// in the system event log; without it the behaviour is unstated.

//

// %s is filled by strArg. Passing the line as the FORMAT string instead would let
// a test label containing a percent sign corrupt the output - or worse.
ADSLOGSTR(msgCtrlMask := Severity OR ADSLOG_MSGTYPE_LOG OR ADSLOG_MSGTYPE_STRING, msgFmtStr := CONCAT(_Prefix, '%s'), strArg := Line);
_LinesWritten := _LinesWritten + 1;
END_METHOD

PROPERTY ErrorsLogged : UDINT
GET
ErrorsLogged := _ErrorsLogged;
END_GET
END_PROPERTY

PROPERTY FailuresLogged : UDINT
GET
FailuresLogged := _FailuresLogged;
END_GET
END_PROPERTY

METHOD FrameworkError
VAR_INPUT
	Source	: T_MaxString;
	Message : T_MaxString;
END_VAR
_FrameworkErrorsLogged := _FrameworkErrorsLogged + 1;

// Always an error, and never silent. This is the framework saying it could not do

// something - a rejected registration, a teardown that overran, a document that

// could not be written - and none of those is a test result.
THIS^.Emit(ADSLOG_MSGTYPE_ERROR, CONCAT(CONCAT('FRAMEWORK ', Source), CONCAT(': ', Message)));
END_METHOD

PROPERTY FrameworkErrorsLogged : UDINT
GET
FrameworkErrorsLogged := _FrameworkErrorsLogged;
END_GET
END_PROPERTY

// Always TRUE. ADSLOGSTR completes within the call, so this sink never holds a

// run open - which is precisely why it is the one to attach first.
PROPERTY IsIdle : BOOL
GET
IsIdle := TRUE;
END_GET
END_PROPERTY

// Every line this sink has written. Assert it in CI if the log is the artifact.
PROPERTY LinesWritten : UDINT
GET
LinesWritten := _LinesWritten;
END_GET
END_PROPERTY

METHOD RunFinished
VAR_INPUT
	Status	   : I_TestRunStatus;
	TargetInfo : T_MaxString;
END_VAR

VAR
	Line : T_MaxString;
END_VAR
IF Status = 0 THEN
	RETURN;
END_IF

// TargetInfo identifies where the run happened. Without it a matrix run across

// several targets produces log output that cannot be told apart.
Line := CONCAT(CONCAT(THIS^.Tally(Status), '  on '), TargetInfo);
THIS^.Emit(ADSLOG_MSGTYPE_HINT, _Rule);
// Severity follows the outcome. A log filtered to errors still shows the closing

// line of a run that went red, and shows nothing of one that did not.
//

// The same four banners, at the same severities, as the suite line. Skipped is

// not red, so it is not logged as an error; Errored is kept apart from Failed

// because nothing about the code was shown, and the reader should look elsewhere.
IF Status.Outcome = E_RunOutcome.Passed THEN
	THIS^.Emit(ADSLOG_MSGTYPE_HINT, CONCAT('===  RUN PASSED  ', Line));
ELSIF Status.Outcome = E_RunOutcome.Skipped THEN
	THIS^.Emit(ADSLOG_MSGTYPE_HINT, CONCAT('===  RUN SKIPPED ', Line));
ELSIF Status.Outcome = E_RunOutcome.Errored THEN
	THIS^.Emit(ADSLOG_MSGTYPE_ERROR, CONCAT('===  RUN ERRORED ', Line));
ELSE
	THIS^.Emit(ADSLOG_MSGTYPE_ERROR, CONCAT('===  RUN FAILED  ', Line));
END_IF

THIS^.Emit(ADSLOG_MSGTYPE_HINT, _Rule);
END_METHOD

// Opens the run with a banner, so everything between it and the closing rule

// belongs to this run and nothing else.

//

// The TwinCAT log is shared - a machine writes to it too - and test output is

// interleaved with whatever else is happening. Without a marker at BOTH ends, a

// reader scrolling back cannot tell where the run began; the failures stream

// during it and the summary only arrives at the end.
METHOD RunStarted
VAR_INPUT
	Label	   : T_MaxString;
	TargetInfo : T_MaxString;
END_VAR

VAR
	Line : T_MaxString;
END_VAR
THIS^.Emit(ADSLOG_MSGTYPE_HINT, _Rule);
Line := CONCAT('===  TEST RUN  ', Label);
IF TargetInfo <> '' THEN
	Line := CONCAT(Line, CONCAT('  on ', TargetInfo));
END_IF

THIS^.Emit(ADSLOG_MSGTYPE_HINT, Line);
THIS^.Emit(ADSLOG_MSGTYPE_HINT, _Rule);
END_METHOD

// Prepended to every line. Useful when several runs share one log - a rig

// running unit and integration suites, or a matrix across targets.
METHOD SetPrefix
VAR_INPUT
	Prefix : T_MaxString;
END_VAR
_Prefix := Prefix;
END_METHOD

// Which results reach the log. Default: failures and errors only.

//

// A suite of eighty passing tests writing eighty log lines buries the two that

// matter. Passes are counted, not narrated - the counts are already available

// through I_TestRunStatus for anyone who wants them.
METHOD SetVerbosity
VAR_INPUT
	// TRUE also logs a line for every passing and skipped test.
	IncludePasses : BOOL;
END_VAR
_IncludePasses := IncludePasses;
END_METHOD

METHOD SuiteFinished
VAR_INPUT
	Status : I_TestRunStatus;
END_VAR

VAR
	Line : T_MaxString;
END_VAR
IF Status = 0 THEN
	RETURN;
END_IF

_SuitesSeen := _SuitesSeen + 1;
Line		:= CONCAT(CONCAT(Status.Label, ': '), THIS^.Tally(Status));
// Severity follows the outcome, so a log filtered to errors still shows which

// suite was responsible rather than only the individual failures.
IF Status.Outcome = E_RunOutcome.Passed THEN
	THIS^.Emit(ADSLOG_MSGTYPE_HINT, CONCAT('SUITE PASSED  ', Line));
ELSIF Status.Outcome = E_RunOutcome.Skipped THEN
	THIS^.Emit(ADSLOG_MSGTYPE_HINT, CONCAT('SUITE SKIPPED ', Line));
ELSIF Status.Outcome = E_RunOutcome.Errored THEN
	THIS^.Emit(ADSLOG_MSGTYPE_ERROR, CONCAT('SUITE ERRORED ', Line));
ELSE
	THIS^.Emit(ADSLOG_MSGTYPE_ERROR, CONCAT('SUITE FAILED  ', Line));
END_IF
END_METHOD

PROPERTY SuitesSeen : UDINT
GET
SuitesSeen := _SuitesSeen;
END_GET
END_PROPERTY

// The counts as one readable phrase. Shared by the suite and run lines so the two

// cannot drift apart.
METHOD Tally : T_MaxString
VAR_INPUT
	Status : I_TestRunStatus;
END_VAR
IF Status = 0 THEN
	RETURN;
END_IF

Tally := CONCAT(UDINT_TO_STRING(Status.PassedCount), ' passed');
Tally := CONCAT(Tally, CONCAT(', ', UDINT_TO_STRING(Status.FailedCount)));
Tally := CONCAT(Tally, ' failed');
Tally := CONCAT(Tally, CONCAT(', ', UDINT_TO_STRING(Status.ErrorCount)));
Tally := CONCAT(Tally, ' errored');
Tally := CONCAT(Tally, CONCAT(', ', UDINT_TO_STRING(Status.SkippedCount)));
Tally := CONCAT(Tally, ' skipped, of ');
Tally := CONCAT(Tally, UDINT_TO_STRING(Status.TestCount));
END_METHOD

METHOD TestFinished
VAR_INPUT
	SuiteLabel	  : T_MaxString;
	TestLabel	  : T_MaxString;
	Location	  : T_MaxString;
	Status		  : E_TestStatus;
	Kind		  : E_FailureKind;
	Summary		  : T_MaxString;
	ElapsedTime	  : LREAL;
	ElapsedCycles : UDINT;
	Assertions	  : UDINT;
END_VAR

VAR
	Line : T_MaxString;
END_VAR
_TestsSeen := _TestsSeen + 1;
CASE Status OF
	E_TestStatus.Failed:
		_FailuresLogged := _FailuresLogged + 1;

		// The summary is already composed to fit one line, kind first in its own field.

		// Repeating the kind here would spend characters the summary needs.
		Line := CONCAT(CONCAT(CONCAT(CONCAT('FAILED ', SuiteLabel), ' / '), TestLabel), CONCAT(': ', Summary));
		THIS^.Emit(ADSLOG_MSGTYPE_ERROR, Line);

	E_TestStatus.Errored:
		_ErrorsLogged := _ErrorsLogged + 1;

		// Warning, not error: the code under test was never shown to be wrong. A build

		// should react differently, and so should whoever is reading the log.
		Line := CONCAT(CONCAT(CONCAT(CONCAT('ERRORED ', SuiteLabel), ' / '), TestLabel), CONCAT(': ', Summary));
		THIS^.Emit(ADSLOG_MSGTYPE_WARN, Line);

	E_TestStatus.Skipped:
		// Narrated only when asked, like a pass - but named for what it is. Sharing
		// the pass branch would write "passed" for a test that never ran.
		IF _IncludePasses THEN
			Line := CONCAT(CONCAT(CONCAT('skipped ', SuiteLabel), ' / '), TestLabel);
			THIS^.Emit(ADSLOG_MSGTYPE_HINT, Line);
		END_IF

ELSE
	IF _IncludePasses THEN
		Line := CONCAT(CONCAT(CONCAT('passed ', SuiteLabel), ' / '), TestLabel);
		THIS^.Emit(ADSLOG_MSGTYPE_HINT, Line);
	END_IF
END_CASE
END_METHOD

// Every test notified, whether or not it produced a line.
PROPERTY TestsSeen : UDINT
GET
TestsSeen := _TestsSeen;
END_GET
END_PROPERTY

END_FUNCTION_BLOCK

// ---- Project Information/F_GetCompany.TcPOU
// This function has been automatically generated from the project information.
{attribute 'signature_flag' := '1073741824'}
{attribute 'TcGenerated'}
{attribute 'no-analysis'}
FUNCTION F_GetCompany : WSTRING
VAR_INPUT
END_VAR

F_GetCompany := "None";

END_FUNCTION

// ---- Project Information/F_GetTitle.TcPOU
// This function has been automatically generated from the project information.
{attribute 'signature_flag' := '1073741824'}
{attribute 'TcGenerated'}
{attribute 'no-analysis'}
FUNCTION F_GetTitle : WSTRING
VAR_INPUT
END_VAR

F_GetTitle := "TestHarnessCore";

END_FUNCTION

// ---- Project Information/F_GetVersion.TcPOU
// This function has been automatically generated from the project information.
{attribute 'signature_flag' := '1073741824'}
{attribute 'TcGenerated'}
{attribute 'no-analysis'}
FUNCTION F_GetVersion : ST_LibVersion
VAR_INPUT
	
END_VAR

F_GetVersion.iMajor := 0;
F_GetVersion.iMinor := 0;
F_GetVersion.iBuild := 11;
F_GetVersion.iRevision := 0;
F_GetVersion.sVersion := '0.0.11';
F_GetVersion.nFlags := 0;

END_FUNCTION
